Yaskawa INFORM job: shotblast_cylinder_program.JBI

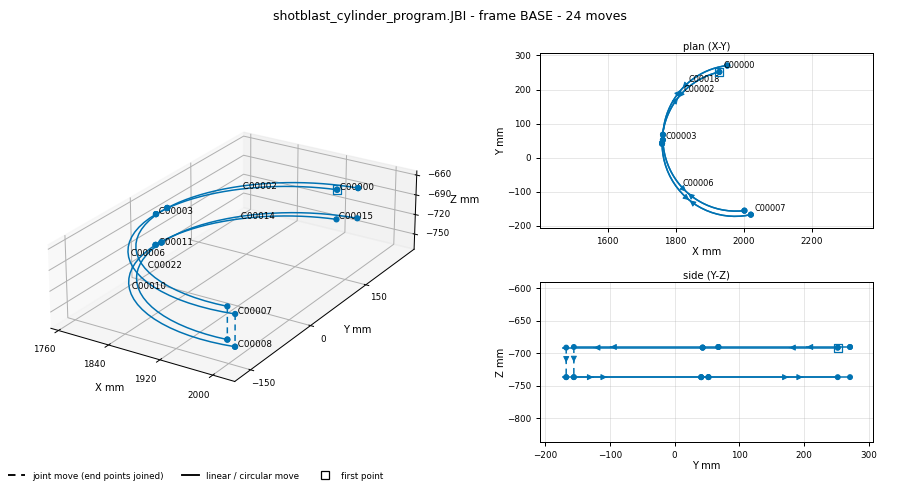
[picture p0: tool path of shotblast_cylinder_program.JBI in frame BASE, 24 of 37 moves have a stored position in this frame; points joined in program order, loops and branches not executed]
/JOB
//NAME shotblast_cylinder_program
//POS
///NPOS 32,0,32,0,0,0
///TOOL 0
///POSTYPE BASE
///RECTAN
///RCONF 0,0,0,0,0,0,0,0,0,0,0,0,0,0,0,0,0,0,0,0,0,0,0,0
C00000=1927.842904,251.570359,-691.250460,175.000000,-60.000000,-77.485875
C00001=1927.842904,251.570359,-691.250460,175.000000,-60.000000,-77.485875
C00002=1810.326308,180.391065,-691.250460,175.000000,-60.000000,-40.107909
C00003=1759.911763,43.262469,-691.250460,175.000000,-60.000000,-5.000000
C00004=1759.911763,43.262469,-691.250460,175.000000,-60.000000,-5.000000
C00005=1759.911763,43.262469,-691.250460,175.000000,-60.000000,-5.000000
C00006=1808.072734,-93.116773,-691.250460,175.000000,-60.000000,39.163750
C00007=2020.476875,-167.077070,-691.250460,-175.000000,-60.000000,102.439450
C00008=2020.285356,-167.119224,-736.836460,175.000000,-60.000000,102.387041
C00009=2020.285356,-167.119224,-736.836460,175.000000,-60.000000,102.387041
C00010=1810.472386,-96.010649,-736.836460,-175.000000,-60.000000,40.168470
C00011=1759.913011,41.049397,-736.836460,175.000000,-60.000000,5.000000
C00012=1759.913011,41.049397,-736.836460,175.000000,-60.000000,5.000000
C00013=1759.913011,41.049397,-736.836460,175.000000,-60.000000,5.000000
C00014=1808.758539,178.508067,-736.836460,-175.000000,-60.000000,-39.453073
C00015=1927.762162,251.552421,-736.836460,175.000000,-60.000000,-77.463771
C00016=1951.181414,270.506131,-690.287460,-175.000000,-60.000000,-83.227022
C00017=1951.181414,270.506131,-690.287460,-175.000000,-60.000000,-83.227022
C00018=1825.401101,209.738199,-690.287460,175.000000,-60.000000,-45.200043
C00019=1762.308148,67.536754,-690.287460,175.000000,-60.000000,-5.000000
C00020=1762.308148,67.536754,-690.287460,175.000000,-60.000000,-5.000000
C00021=1762.308148,67.536754,-690.287460,175.000000,-60.000000,-5.000000
C00022=1849.405653,-115.062124,-690.287460,-175.000000,-60.000000,53.653629
C00023=2001.560310,-155.297499,-690.287460,175.000000,-60.000000,96.722169
C00024=2001.398414,-155.316518,-736.784460,-175.000000,-60.000000,96.678605
C00025=2001.398414,-155.316518,-736.784460,-175.000000,-60.000000,96.678605
C00026=1810.237564,-77.773042,-736.784460,175.000000,-60.000000,39.162001
C00027=1762.145993,52.234763,-736.784460,175.000000,-60.000000,5.000000
C00028=1762.145993,52.234763,-736.784460,175.000000,-60.000000,5.000000
C00029=1762.145993,52.234763,-736.784460,175.000000,-60.000000,5.000000
C00030=1820.348313,204.548119,-736.784460,175.000000,-60.000000,-43.264108
C00031=1951.125788,270.499517,-736.784460,-175.000000,-60.000000,-83.212051
///POSTYPE PULSE
///PULSE
EX00000=104448.0
EX00001=283648.0
///POSTYPE PULSE
///PULSE
EC00000=104448.0
EC00001=104448.0
EC00002=104448.0
EC00003=104448.0
EC00004=104448.0
EC00005=104448.0
EC00006=104448.0
EC00007=104448.0
EC00008=104448.0
EC00009=104448.0
EC00010=104448.0
EC00011=104448.0
EC00012=104448.0
EC00013=104448.0
EC00014=104448.0
EC00015=104448.0
EC00016=283648.0
EC00017=283648.0
EC00018=283648.0
EC00019=283648.0
EC00020=283648.0
EC00021=283648.0
EC00022=283648.0
EC00023=283648.0
EC00024=283648.0
EC00025=283648.0
EC00026=283648.0
EC00027=283648.0
EC00028=283648.0
EC00029=283648.0
EC00030=283648.0
EC00031=283648.0
//INST
///DATE 2023/08/16 11:59
///ATTR SC,RW,RJ
////FRAME BASE
///GROUP1 RB1,ST1
NOP
MOVJ P009 EX000 VJ=15.00
MOVJ C00000 EC00000 VJ=15.0
CALL JOB:SPYON
MOVC C00001 EC00001 V=150.0
MOVC C00002 EC00002 V=150.0
MOVC C00003 EC00003 V=150.0
MOVJ C00004 EC00004 VJ=15.0
MOVC C00005 EC00005 V=150.0
MOVC C00006 EC00006 V=150.0
MOVC C00007 EC00007 V=150.0
MOVJ C00008 EC00008 VJ=15.0
MOVC C00009 EC00009 V=150.0
MOVC C00010 EC00010 V=150.0
MOVC C00011 EC00011 V=150.0
MOVJ C00012 EC00012 VJ=15.0
MOVC C00013 EC00013 V=150.0
MOVC C00014 EC00014 V=150.0
MOVC C00015 EC00015 V=150.0
CALL JOB:SPYOF
MOVJ P009 VJ=15.00
MOVL P009 EX00000 V=150.0
MOVJ C00016 EC00016 VJ=15.0
CALL JOB:SPYON
MOVC C00017 EC00017 V=150.0
MOVC C00018 EC00018 V=150.0
MOVC C00019 EC00019 V=150.0
MOVJ C00020 EC00020 VJ=15.0
MOVC C00021 EC00021 V=150.0
MOVC C00022 EC00022 V=150.0
MOVC C00023 EC00023 V=150.0
MOVJ C00024 EC00024 VJ=15.0
MOVC C00025 EC00025 V=150.0
MOVC C00026 EC00026 V=150.0
MOVC C00027 EC00027 V=150.0
MOVJ C00028 EC00028 VJ=15.0
MOVC C00029 EC00029 V=150.0
MOVC C00030 EC00030 V=150.0
MOVC C00031 EC00031 V=150.0
CALL JOB:SPYOF
MOVJ P009 VJ=15.00
MOVL P009 EX00001 V=150.0
END
